{attribute 'GeneratedUsingTerminal: EJ5151-0000-0016'}
{attribute addProperty BoxType "EJ5151-0000-0016"}
{attribute addProperty Id "ControlAT %Q*Control_6EF2C5D04Set_counter_valueAT %Q*UINT2"}
{attribute addProperty CRC "568512845"}
{attribute addProperty Size "6"}
TYPE ENC_Outputs_21E2D14D EXTENDS OutputBase_10CEE7DE :
STRUCT
	{attribute addProperty Name "Control"}
	Control AT %Q* : Control_6EF2C5D0;
	{attribute addProperty Name "Set_counter_value"}
	Set_counter_value AT %Q* : UINT;
END_STRUCT
END_TYPE

(* stored: Version 1.2.0.0, ProductVersion 3.1.4024.9
   DUT ENC_Outputs_21E2D14D: Id {e51003e2-3059-44b0-8c77-7458d3b54f06} *)
